// TIA Portal V16 export
// export: Created 2021-11-12T13:31:16.9009323Z, ExportSetting WithDefaults, DisplayName Totally Integrated Automation Portal, DisplayVersion V16 Update 3, DisplayName TIA Portal Version Control Interface, DisplayVersion V16 Update 2, DisplayName TIA Portal Openness, DisplayVersion V16 Update 3, DisplayName SINAMICS Startdrive Advanced, DisplayVersion V16 Update 5, DisplayName SINAMICS Startdrive G130, G150, S120, S150, SINAMICS MV, S210, DisplayVersion V16 Update 5, DisplayName SINAMICS Startdrive G110M, G120, G120C, G120D, G120P, G115D, DisplayVersion V16 Update 5, DisplayName STEP 7 Professional, DisplayVersion V16 Update 3, DisplayName STEP 7 Safety, DisplayVersion V16, DisplayName WinCC UA Professional, DisplayVersion V16 Update 3
FUNCTION_BLOCK "STD_Station"   // FB1101, LAD
TITLE = STD_Station
{ S7_Optimized_Access := 'TRUE' }
VERSION : 0.1
// Control of station - part of zone
// stored: AutoNumber false, IsIECCheckEnabled false, IsRetainMemResEnabled false, MemoryReserve 100, SetENOAutomatically false, UDAEnableTagReadback false
   VAR_INPUT
      IS_ZoneM : "UDT_Status_main";   // Status of zone
      IS_ZoneS : "UDT_Zone_Status_specific";   // Status of zone
      IB1StnExtCtrl : Bool;   // External control of station - own logic for automatic run
      IB1StnAutoRun : Bool;   // Station in automatic run mode - external signal
      IB1Rmt : Bool;   // Remote operation - operation from HMI panel
      IB1ManSwch : Bool;   // Switch in manual position
      IB1AutSwch : Bool;   // Switch in automatic position
      IB1SftyOK : Bool;   // Safety circuits ON
      IB1Run : Bool;   // Any device running
      IB1CollWrn : Bool;   // Any warning evaluated
      IB1CollErr : Bool;   // Any error evaluated
      IB1AllAutoRun : Bool;   // All drives in automatic run mode
      IB1AllEndOfCycle : Bool;   // All devices in end of cycle
      IB1AllEndOfProd : Bool;   // Production finished on all devices
      IB1AllInBasePos : Bool;   // All stations in base position
      IB1AllStopBefor : Bool;   // All stations stopped before operation
      IB1AllStopAfter : Bool;   // All stations stopped after finishing of operation
      IB1ReqBasePos : Bool;   // Request to move devices to base position
      IB1ReqEndOfCycle : Bool;   // Request for end of cycle
      IB1ReqEndOfProdAct : Bool;   // Request for end of production selection
      IB1ReqEndOfProdCncl : Bool;   // Request for end of production deselection
      IB1AutStartBtn : Bool;   // Button to start automatic
      IB1Stop : Bool;   // Command stop
      IB1Blink : Bool;   // Pulses for blinking
      IB1AlmSupp : Bool;   // Alarms suppressed
      II_DevSelNr : Int;   // Number of selected devices
   END_VAR
   VAR_OUTPUT
      OS_Status : Struct   // Output status
         Main : "UDT_Status_main";
         Specific : "UDT_Zone_Status_specific";
         Error : "UDT_Error01";
      END_STRUCT;
      OB1AutStart : Bool;   // LED for automatic start button
      OB1Man : Bool;   // LED for manual mode signalisation
      OB1Rmt : Bool;   // LED for remote control signalisation
      OB1SigAcs : Bool;   // Acoustic signalisation
   END_VAR
   VAR_IN_OUT
      XS_Parameter : "UDT_Station_Parameter";   // Parameters
      XS_Command : "UDT_Station_Command";   // Commands
   END_VAR
   VAR
      SS_Alarm : Struct   // Zone alarms
         Res_0_0 : Bool;
         Res_0_1 : Bool;
         Res_0_2 : Bool;
         Res_0_3 : Bool;
         Res_0_4 : Bool;
         Res_0_5 : Bool;
         Res_0_6 : Bool;
         Res_0_7 : Bool;
      END_STRUCT;
      SS_Warning : Struct   // Zone warnings
         EndOfCycle : Bool;   // End of cycle mode active / Konec cyklu aktivní / Mode de fin de cycle actif
         EndOfProd : Bool;   // End of production mode active / Konec produkce aktivní / Fin du mode de production actif
         StepMode : Bool;   // Step mode active / Krokový automat aktivní / Mode pas à pas actif
         StopBefor : Bool;   // Stop before operation active / Zastavení před procesem aktivní / Arrêtez avant l'opération actif
         StopAfter : Bool;   // Stop after operation active / Zastavení po procesu aktivní / Arrêter après l'opération actif
         BypasMode : Bool;   // Bypass mode active / Vynechání procesu aktivní / Mode bypass actif
         Res_0_6 : Bool;
         Res_0_7 : Bool;
      END_STRUCT;
      SB1AutoRun : Bool;   // Automatic operation started
      SB1AutoRunBasePos : Bool;   // Automatic operation - Run to base position
      SB1AutoRunProd : Bool;   // Automatic operation - Production
      SB1ModeAutStep : Bool;   // Mode automatic step selected
      SB1ModeStopBefor : Bool;   // Mode stop before production saelected
      SB1ModeStopAfter : Bool;   // Mode stop after production selected
      SB1ModeBypas : Bool;   // Mode bypass selected
      SB1ModeAut : Bool;   // Mode automatic
      SB1ModeMan : Bool;   // Mode manual
      SB1ModeOff : Bool;   // Mode off
      SB1ReqEndOfCycle : Bool;   // Request for end of cycle
      SB1ReqEndOfProd : Bool;   // Request for end of production
      SB1ManAutPE : Bool;   // Manual mode - positive edge
      SB1OffPE : Bool;   // Off mode - positive edge
      SB1ReqBasePosPE : Bool;   // Request for base position - positive edge
      SB1ReqEndOfCyclePE : Bool;   // Request end of cycle - positive edge
      SB1ReqEndOfProdActPE : Bool;   // Request end of production activation - positive edge
      SB1ReqEndOfProdCnclPE : Bool;   // Request end of production deactivation - positive edge
      SB1AutStart : Bool;   // Pulse start automatic sequence
      SB1AutStartAux : Bool;   // Auxiliary for start sequence
      SB1AuxHorn : Bool;   // To activate Horn before start
      SB1AutStartBtnPE : Bool;   // Automatic start 1 - positive edge
      ST_Horn { S7_SetPoint := 'True'} : TON_TIME;   // Timer for horn
      ST_Start { S7_SetPoint := 'True'} : TON_TIME;   // Timer to activate horn before start
      ST_AlmSupp { S7_SetPoint := 'True'} : IEC_TIMER;
   END_VAR
   VAR_TEMP
      TS_Status : Struct
         Main : "UDT_Status_main";
         Specific : "UDT_Zone_Status_specific";
         Error : "UDT_Error01";
      END_STRUCT;
      TS_Parameter : "UDT_Station_Parameter";   // Parameters
      TS_Command : "UDT_Station_Command";   // Commands
      TB1AlmSupp : Bool;
      TB1CollWrn : Bool;
      TB1ReqBasePosPE : Bool;   // Request for base position - positive edge
      TB1ReqEndOfCyclePE : Bool;   // Request end of cycle - positive edge
      TB1ReqEndOfProdActPE : Bool;   // Request end of production activation - positive edge
      TB1ReqEndOfProdCnclPE : Bool;   // Request end of production deactivation - positive edge
      TB1SigHorn : Bool;   // Horn before start signalisation
      TB1AutStartBtnPE : Bool;   // Automatic start 1 - positive edge
   END_VAR
   VAR CONSTANT
      CT_Horn : Time := T#2s;   // Time for horn before start
      CT_Start : Time := T#1s;   // Time for delay before start
      CT_AlmSupp : Time := T#3s;   // Time to delay alarm release
   END_VAR
   VAR_TEMP   // added for the SCL form of the ladder/FBD networks
      _w1 : Bool;
      _w2 : Bool;
   END_VAR
BEGIN

REGION Network 1: Clear temporary variables TS_Status - Main, Specific
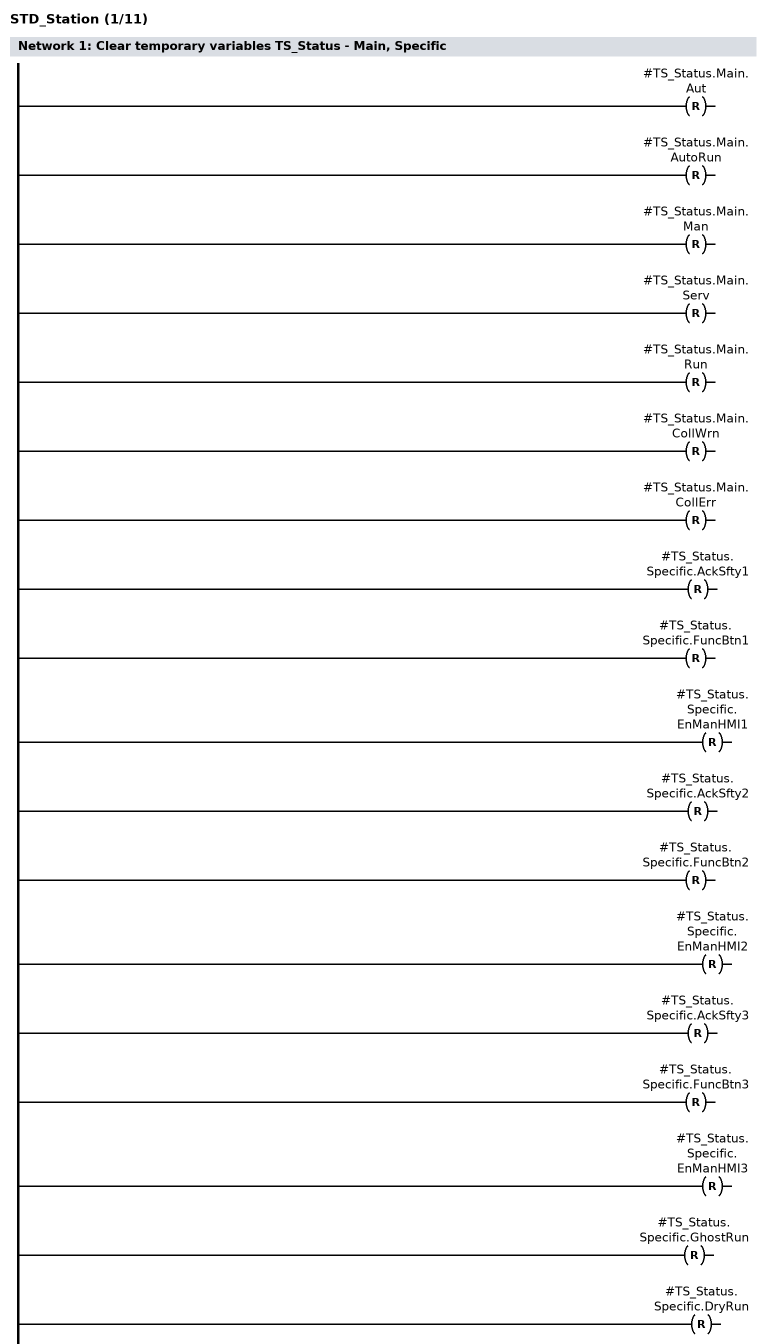
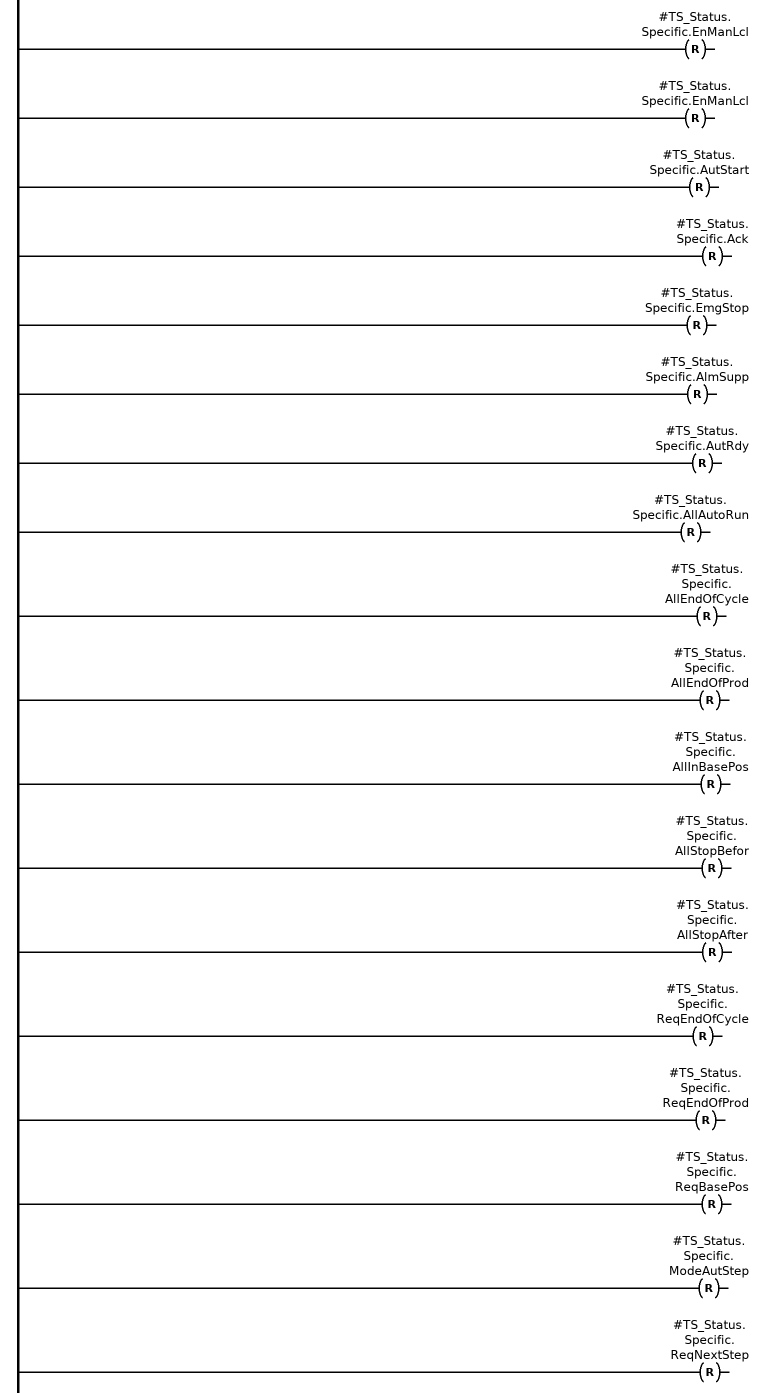
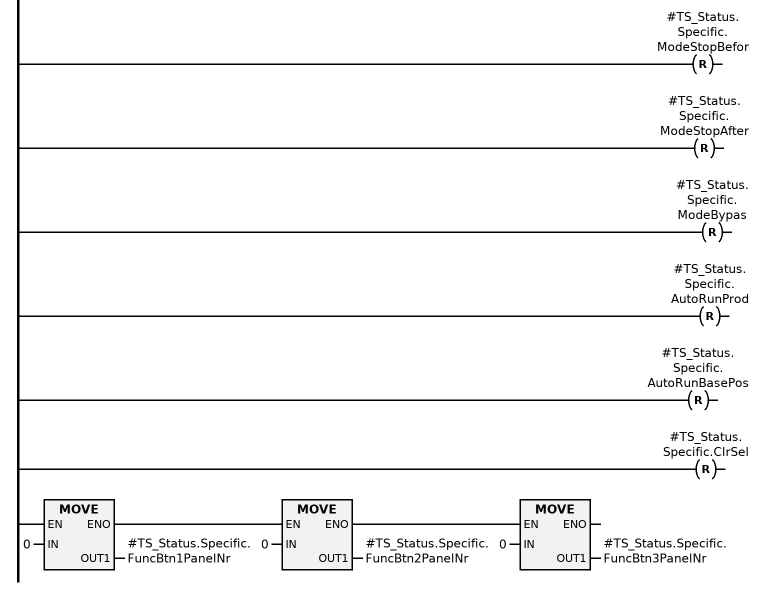
   RUNG wire#powerrail
      R_Coil( #TS_Status.Main.Aut )
   END_RUNG
   RUNG wire#powerrail
      R_Coil( #TS_Status.Main.AutoRun )
   END_RUNG
   RUNG wire#powerrail
      R_Coil( #TS_Status.Main.Man )
   END_RUNG
   RUNG wire#powerrail
      R_Coil( #TS_Status.Main.Serv )
   END_RUNG
   RUNG wire#powerrail
      R_Coil( #TS_Status.Main.Run )
   END_RUNG
   RUNG wire#powerrail
      R_Coil( #TS_Status.Main.CollWrn )
   END_RUNG
   RUNG wire#powerrail
      R_Coil( #TS_Status.Main.CollErr )
   END_RUNG
   RUNG wire#powerrail
      R_Coil( #TS_Status.Specific.AckSfty1 )
   END_RUNG
   RUNG wire#powerrail
      R_Coil( #TS_Status.Specific.FuncBtn1 )
   END_RUNG
   RUNG wire#powerrail
      R_Coil( #TS_Status.Specific.EnManHMI1 )
   END_RUNG
   RUNG wire#powerrail
      R_Coil( #TS_Status.Specific.AckSfty2 )
   END_RUNG
   RUNG wire#powerrail
      R_Coil( #TS_Status.Specific.FuncBtn2 )
   END_RUNG
   RUNG wire#powerrail
      R_Coil( #TS_Status.Specific.EnManHMI2 )
   END_RUNG
   RUNG wire#powerrail
      R_Coil( #TS_Status.Specific.AckSfty3 )
   END_RUNG
   RUNG wire#powerrail
      R_Coil( #TS_Status.Specific.FuncBtn3 )
   END_RUNG
   RUNG wire#powerrail
      R_Coil( #TS_Status.Specific.EnManHMI3 )
   END_RUNG
   RUNG wire#powerrail
      R_Coil( #TS_Status.Specific.GhostRun )
   END_RUNG
   RUNG wire#powerrail
      R_Coil( #TS_Status.Specific.DryRun )
   END_RUNG
   RUNG wire#powerrail
      R_Coil( #TS_Status.Specific.EnManLcl )
   END_RUNG
   RUNG wire#powerrail
      R_Coil( #TS_Status.Specific.EnManLcl )
   END_RUNG
   RUNG wire#powerrail
      R_Coil( #TS_Status.Specific.AutStart )
   END_RUNG
   RUNG wire#powerrail
      R_Coil( #TS_Status.Specific.Ack )
   END_RUNG
   RUNG wire#powerrail
      R_Coil( #TS_Status.Specific.EmgStop )
   END_RUNG
   RUNG wire#powerrail
      R_Coil( #TS_Status.Specific.AlmSupp )
   END_RUNG
   RUNG wire#powerrail
      R_Coil( #TS_Status.Specific.AutRdy )
   END_RUNG
   RUNG wire#powerrail
      R_Coil( #TS_Status.Specific.AllAutoRun )
   END_RUNG
   RUNG wire#powerrail
      R_Coil( #TS_Status.Specific.AllEndOfCycle )
   END_RUNG
   RUNG wire#powerrail
      R_Coil( #TS_Status.Specific.AllEndOfProd )
   END_RUNG
   RUNG wire#powerrail
      R_Coil( #TS_Status.Specific.AllInBasePos )
   END_RUNG
   RUNG wire#powerrail
      R_Coil( #TS_Status.Specific.AllStopBefor )
   END_RUNG
   RUNG wire#powerrail
      R_Coil( #TS_Status.Specific.AllStopAfter )
   END_RUNG
   RUNG wire#powerrail
      R_Coil( #TS_Status.Specific.ReqEndOfCycle )
   END_RUNG
   RUNG wire#powerrail
      R_Coil( #TS_Status.Specific.ReqEndOfProd )
   END_RUNG
   RUNG wire#powerrail
      R_Coil( #TS_Status.Specific.ReqBasePos )
   END_RUNG
   RUNG wire#powerrail
      R_Coil( #TS_Status.Specific.ModeAutStep )
   END_RUNG
   RUNG wire#powerrail
      R_Coil( #TS_Status.Specific.ReqNextStep )
   END_RUNG
   RUNG wire#powerrail
      R_Coil( #TS_Status.Specific.ModeStopBefor )
   END_RUNG
   RUNG wire#powerrail
      R_Coil( #TS_Status.Specific.ModeStopAfter )
   END_RUNG
   RUNG wire#powerrail
      R_Coil( #TS_Status.Specific.ModeBypas )
   END_RUNG
   RUNG wire#powerrail
      R_Coil( #TS_Status.Specific.AutoRunProd )
   END_RUNG
   RUNG wire#powerrail
      R_Coil( #TS_Status.Specific.AutoRunBasePos )
   END_RUNG
   RUNG wire#powerrail
      R_Coil( #TS_Status.Specific.ClrSel )
   END_RUNG
   RUNG wire#powerrail
      { S7_GenerateENO := "TRUE" } Move(in := 0, out1 => #TS_Status.Specific.FuncBtn1PanelNr)
      { S7_GenerateENO := "TRUE" } Move(in := 0, out1 => #TS_Status.Specific.FuncBtn2PanelNr)
      { S7_GenerateENO := "TRUE" } Move(in := 0, out1 => #TS_Status.Specific.FuncBtn3PanelNr)
   END_RUNG
   // the same network as SCL:
   // ENO of a box is taken as its EN; it also drops when the box reports an error
   #TS_Status.Main.Aut := FALSE;
   #TS_Status.Main.AutoRun := FALSE;
   #TS_Status.Main.Man := FALSE;
   #TS_Status.Main.Serv := FALSE;
   #TS_Status.Main.Run := FALSE;
   #TS_Status.Main.CollWrn := FALSE;
   #TS_Status.Main.CollErr := FALSE;
   #TS_Status.Specific.AckSfty1 := FALSE;
   #TS_Status.Specific.FuncBtn1 := FALSE;
   #TS_Status.Specific.EnManHMI1 := FALSE;
   #TS_Status.Specific.AckSfty2 := FALSE;
   #TS_Status.Specific.FuncBtn2 := FALSE;
   #TS_Status.Specific.EnManHMI2 := FALSE;
   #TS_Status.Specific.AckSfty3 := FALSE;
   #TS_Status.Specific.FuncBtn3 := FALSE;
   #TS_Status.Specific.EnManHMI3 := FALSE;
   #TS_Status.Specific.GhostRun := FALSE;
   #TS_Status.Specific.DryRun := FALSE;
   #TS_Status.Specific.EnManLcl := FALSE;
   #TS_Status.Specific.EnManLcl := FALSE;
   #TS_Status.Specific.AutStart := FALSE;
   #TS_Status.Specific.Ack := FALSE;
   #TS_Status.Specific.EmgStop := FALSE;
   #TS_Status.Specific.AlmSupp := FALSE;
   #TS_Status.Specific.AutRdy := FALSE;
   #TS_Status.Specific.AllAutoRun := FALSE;
   #TS_Status.Specific.AllEndOfCycle := FALSE;
   #TS_Status.Specific.AllEndOfProd := FALSE;
   #TS_Status.Specific.AllInBasePos := FALSE;
   #TS_Status.Specific.AllStopBefor := FALSE;
   #TS_Status.Specific.AllStopAfter := FALSE;
   #TS_Status.Specific.ReqEndOfCycle := FALSE;
   #TS_Status.Specific.ReqEndOfProd := FALSE;
   #TS_Status.Specific.ReqBasePos := FALSE;
   #TS_Status.Specific.ModeAutStep := FALSE;
   #TS_Status.Specific.ReqNextStep := FALSE;
   #TS_Status.Specific.ModeStopBefor := FALSE;
   #TS_Status.Specific.ModeStopAfter := FALSE;
   #TS_Status.Specific.ModeBypas := FALSE;
   #TS_Status.Specific.AutoRunProd := FALSE;
   #TS_Status.Specific.AutoRunBasePos := FALSE;
   #TS_Status.Specific.ClrSel := FALSE;
   #TS_Status.Specific.FuncBtn1PanelNr := 0;
   #TS_Status.Specific.FuncBtn2PanelNr := 0;
   #TS_Status.Specific.FuncBtn3PanelNr := 0;
END_REGION

REGION Network 2: Copy In/Out variables to temporary variables
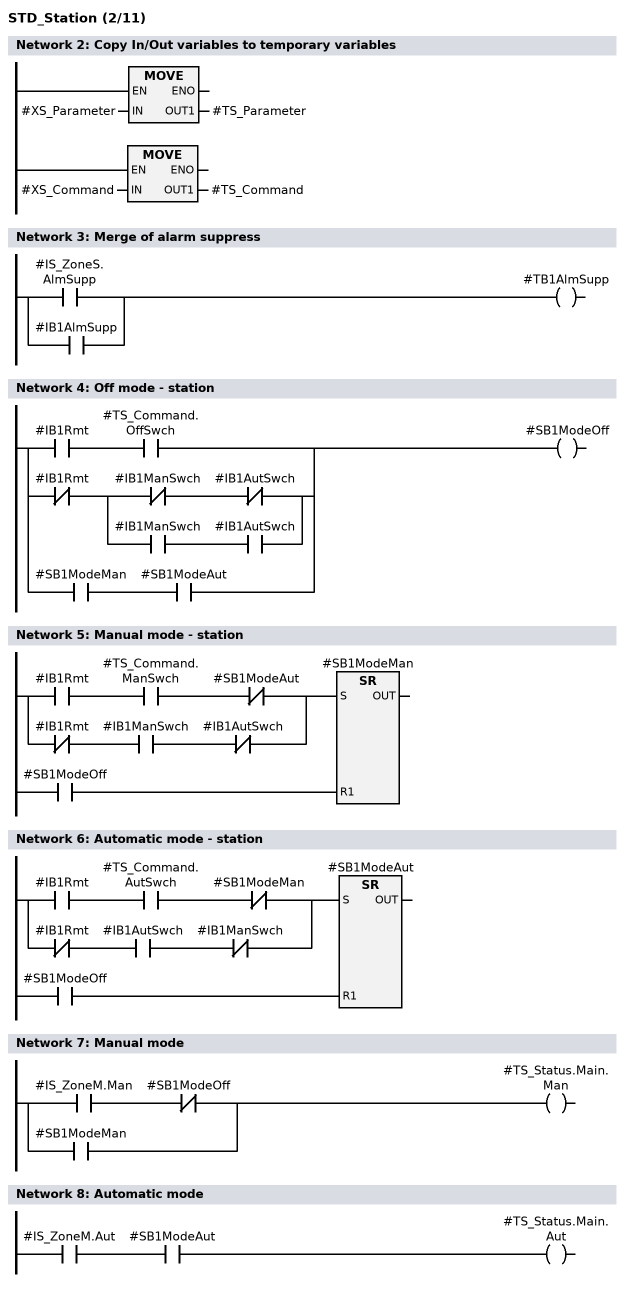
   RUNG wire#powerrail
      { S7_GenerateENO := "TRUE" } Move(in := #XS_Parameter, out1 => #TS_Parameter)
   END_RUNG
   RUNG wire#powerrail
      { S7_GenerateENO := "TRUE" } Move(in := #XS_Command, out1 => #TS_Command)
   END_RUNG
   // the same network as SCL:
   #TS_Parameter := #XS_Parameter;
   #TS_Command := #XS_Command;
END_REGION

REGION Network 3: Merge of alarm suppress
   RUNG wire#powerrail
      Contact( #IS_ZoneS.AlmSupp )
      wire#w1
      Coil( #TB1AlmSupp )
   END_RUNG
   RUNG wire#powerrail
      Contact( #IB1AlmSupp )
   END_RUNG wire#w1
   // the same network as SCL:
   #TB1AlmSupp := #IS_ZoneS.AlmSupp OR #IB1AlmSupp;
END_REGION

REGION Network 4: Off mode - station
   RUNG wire#powerrail
      Contact( #IB1Rmt )
      Contact( #TS_Command.OffSwch )
      wire#w1
      Coil( #SB1ModeOff )
   END_RUNG
   RUNG wire#powerrail
      I_Contact( #IB1Rmt )
      wire#w2
      I_Contact( #IB1ManSwch )
      I_Contact( #IB1AutSwch )
   END_RUNG wire#w1
   RUNG wire#w2
      Contact( #IB1ManSwch )
      Contact( #IB1AutSwch )
   END_RUNG wire#w1
   RUNG wire#powerrail
      Contact( #SB1ModeMan )
      Contact( #SB1ModeAut )
   END_RUNG wire#w1
   // the same network as SCL:
   #SB1ModeOff := (#IB1Rmt AND #TS_Command.OffSwch) OR (NOT #IB1Rmt AND ((NOT #IB1ManSwch AND NOT #IB1AutSwch) OR (#IB1ManSwch AND #IB1AutSwch))) OR (#SB1ModeMan AND #SB1ModeAut);
END_REGION

REGION Network 5: Manual mode - station
   RUNG wire#powerrail
      Contact( #IB1Rmt )
      Contact( #TS_Command.ManSwch )
      I_Contact( #SB1ModeAut )
      wire#w1
      S_SR(operand := #SB1ModeMan, r1 := wire#w2)
   END_RUNG
   RUNG wire#powerrail
      I_Contact( #IB1Rmt )
      Contact( #IB1ManSwch )
      I_Contact( #IB1AutSwch )
   END_RUNG wire#w1
   RUNG wire#powerrail
      Contact( #SB1ModeOff )
   END_RUNG wire#w2
   // the same network as SCL:
   IF (#IB1Rmt AND #TS_Command.ManSwch AND NOT #SB1ModeAut) OR (NOT #IB1Rmt AND #IB1ManSwch AND NOT #IB1AutSwch) THEN
       #SB1ModeMan := TRUE;   // SR flip-flop
   END_IF;
   IF #SB1ModeOff THEN #SB1ModeMan := FALSE; END_IF;
END_REGION

REGION Network 6: Automatic mode - station
   RUNG wire#powerrail
      Contact( #IB1Rmt )
      Contact( #TS_Command.AutSwch )
      I_Contact( #SB1ModeMan )
      wire#w1
      S_SR(operand := #SB1ModeAut, r1 := wire#w2)
   END_RUNG
   RUNG wire#powerrail
      I_Contact( #IB1Rmt )
      Contact( #IB1AutSwch )
      I_Contact( #IB1ManSwch )
   END_RUNG wire#w1
   RUNG wire#powerrail
      Contact( #SB1ModeOff )
   END_RUNG wire#w2
   // the same network as SCL:
   IF (#IB1Rmt AND #TS_Command.AutSwch AND NOT #SB1ModeMan) OR (NOT #IB1Rmt AND #IB1AutSwch AND NOT #IB1ManSwch) THEN
       #SB1ModeAut := TRUE;   // SR flip-flop
   END_IF;
   IF #SB1ModeOff THEN #SB1ModeAut := FALSE; END_IF;
END_REGION

REGION Network 7: Manual mode
   RUNG wire#powerrail
      Contact( #IS_ZoneM.Man )
      I_Contact( #SB1ModeOff )
      wire#w1
      Coil( #TS_Status.Main.Man )
   END_RUNG
   RUNG wire#powerrail
      Contact( #SB1ModeMan )
   END_RUNG wire#w1
   // the same network as SCL:
   #TS_Status.Main.Man := (#IS_ZoneM.Man AND NOT #SB1ModeOff) OR #SB1ModeMan;
END_REGION

REGION Network 8: Automatic mode
   RUNG wire#powerrail
      Contact( #IS_ZoneM.Aut )
      Contact( #SB1ModeAut )
      Coil( #TS_Status.Main.Aut )
   END_RUNG
   // the same network as SCL:
   #TS_Status.Main.Aut := #IS_ZoneM.Aut AND #SB1ModeAut;
END_REGION

REGION Network 9: Automatic start - pulse
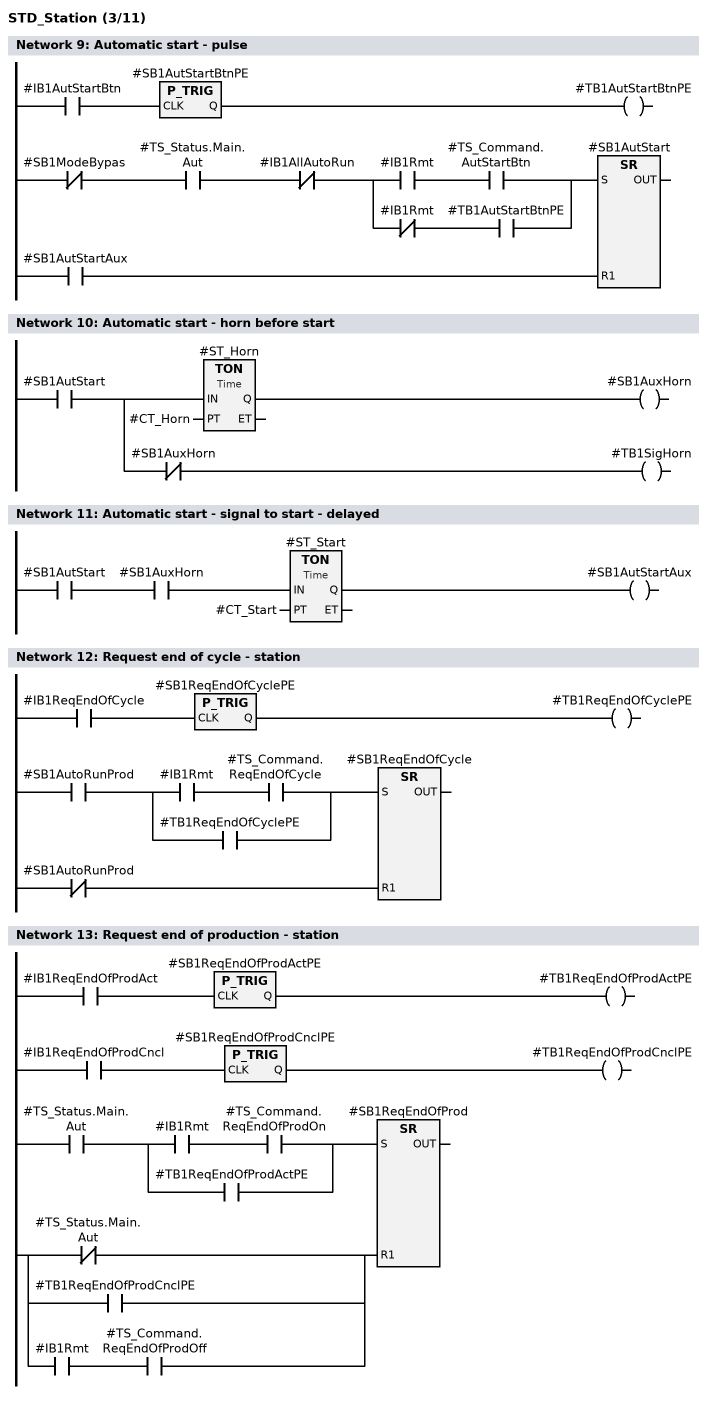
   RUNG wire#powerrail
      Contact( #IB1AutStartBtn )
      P_Trig( #SB1AutStartBtnPE )
      Coil( #TB1AutStartBtnPE )
   END_RUNG
   RUNG wire#powerrail
      I_Contact( #SB1ModeBypas )
      Contact( #TS_Status.Main.Aut )
      I_Contact( #IB1AllAutoRun )
      wire#w1
      Contact( #IB1Rmt )
      Contact( #TS_Command.AutStartBtn )
      wire#w2
      S_SR(operand := #SB1AutStart, r1 := wire#w3)
   END_RUNG
   RUNG wire#w1
      I_Contact( #IB1Rmt )
      Contact( #TB1AutStartBtnPE )
   END_RUNG wire#w2
   RUNG wire#powerrail
      Contact( #SB1AutStartAux )
   END_RUNG wire#w3
   // the same network as SCL:
   #_w1 := #IB1AutStartBtn AND NOT #SB1AutStartBtnPE;   // rising edge
   #SB1AutStartBtnPE := #IB1AutStartBtn;
   #TB1AutStartBtnPE := #_w1;
   IF NOT #SB1ModeBypas AND #TS_Status.Main.Aut AND NOT #IB1AllAutoRun AND ((#IB1Rmt AND #TS_Command.AutStartBtn) OR (NOT #IB1Rmt AND #TB1AutStartBtnPE)) THEN
       #SB1AutStart := TRUE;   // SR flip-flop
   END_IF;
   IF #SB1AutStartAux THEN #SB1AutStart := FALSE; END_IF;
END_REGION

REGION Network 10: Automatic start - horn before start
   RUNG wire#powerrail
      Contact( #SB1AutStart )
      wire#w1
      { S7_Templates := "time_type := Time" } #ST_Horn.TON(pt := #CT_Horn, et =>)
      Coil( #SB1AuxHorn )
   END_RUNG
   RUNG wire#w1
      I_Contact( #SB1AuxHorn )
      Coil( #TB1SigHorn )
   END_RUNG
   // the same network as SCL:
   #ST_Horn(IN := #SB1AutStart, PT := #CT_Horn);   // TON
   #SB1AuxHorn := #ST_Horn.Q;
   #TB1SigHorn := #SB1AutStart AND NOT #SB1AuxHorn;
END_REGION

REGION Network 11: Automatic start - signal to start - delayed
   RUNG wire#powerrail
      Contact( #SB1AutStart )
      Contact( #SB1AuxHorn )
      { S7_Templates := "time_type := Time" } #ST_Start.TON(pt := #CT_Start, et =>)
      Coil( #SB1AutStartAux )
   END_RUNG
   // the same network as SCL:
   #ST_Start(IN := #SB1AutStart AND #SB1AuxHorn, PT := #CT_Start);   // TON
   #SB1AutStartAux := #ST_Start.Q;
END_REGION

REGION Network 12: Request end of cycle - station
   RUNG wire#powerrail
      Contact( #IB1ReqEndOfCycle )
      P_Trig( #SB1ReqEndOfCyclePE )
      Coil( #TB1ReqEndOfCyclePE )
   END_RUNG
   RUNG wire#powerrail
      Contact( #SB1AutoRunProd )
      wire#w1
      Contact( #IB1Rmt )
      Contact( #TS_Command.ReqEndOfCycle )
      wire#w2
      S_SR(operand := #SB1ReqEndOfCycle, r1 := wire#w3)
   END_RUNG
   RUNG wire#w1
      Contact( #TB1ReqEndOfCyclePE )
   END_RUNG wire#w2
   RUNG wire#powerrail
      I_Contact( #SB1AutoRunProd )
   END_RUNG wire#w3
   // the same network as SCL:
   #_w1 := #IB1ReqEndOfCycle AND NOT #SB1ReqEndOfCyclePE;   // rising edge
   #SB1ReqEndOfCyclePE := #IB1ReqEndOfCycle;
   #TB1ReqEndOfCyclePE := #_w1;
   IF #SB1AutoRunProd AND ((#IB1Rmt AND #TS_Command.ReqEndOfCycle) OR #TB1ReqEndOfCyclePE) THEN
       #SB1ReqEndOfCycle := TRUE;   // SR flip-flop
   END_IF;
   IF NOT #SB1AutoRunProd THEN #SB1ReqEndOfCycle := FALSE; END_IF;
END_REGION

REGION Network 13: Request end of production - station
   RUNG wire#powerrail
      Contact( #IB1ReqEndOfProdAct )
      P_Trig( #SB1ReqEndOfProdActPE )
      Coil( #TB1ReqEndOfProdActPE )
   END_RUNG
   RUNG wire#powerrail
      Contact( #IB1ReqEndOfProdCncl )
      P_Trig( #SB1ReqEndOfProdCnclPE )
      Coil( #TB1ReqEndOfProdCnclPE )
   END_RUNG
   RUNG wire#powerrail
      Contact( #TS_Status.Main.Aut )
      wire#w1
      Contact( #IB1Rmt )
      Contact( #TS_Command.ReqEndOfProdOn )
      wire#w2
      S_SR(operand := #SB1ReqEndOfProd, r1 := wire#w3)
   END_RUNG
   RUNG wire#w1
      Contact( #TB1ReqEndOfProdActPE )
   END_RUNG wire#w2
   RUNG wire#powerrail
      I_Contact( #TS_Status.Main.Aut )
   END_RUNG wire#w3
   RUNG wire#powerrail
      Contact( #TB1ReqEndOfProdCnclPE )
   END_RUNG wire#w3
   RUNG wire#powerrail
      Contact( #IB1Rmt )
      Contact( #TS_Command.ReqEndOfProdOff )
   END_RUNG wire#w3
   // the same network as SCL:
   #_w1 := #IB1ReqEndOfProdAct AND NOT #SB1ReqEndOfProdActPE;   // rising edge
   #SB1ReqEndOfProdActPE := #IB1ReqEndOfProdAct;
   #TB1ReqEndOfProdActPE := #_w1;
   #_w2 := #IB1ReqEndOfProdCncl AND NOT #SB1ReqEndOfProdCnclPE;   // rising edge
   #SB1ReqEndOfProdCnclPE := #IB1ReqEndOfProdCncl;
   #TB1ReqEndOfProdCnclPE := #_w2;
   IF #TS_Status.Main.Aut AND ((#IB1Rmt AND #TS_Command.ReqEndOfProdOn) OR #TB1ReqEndOfProdActPE) THEN
       #SB1ReqEndOfProd := TRUE;   // SR flip-flop
   END_IF;
   IF NOT #TS_Status.Main.Aut OR #TB1ReqEndOfProdCnclPE OR (#IB1Rmt AND #TS_Command.ReqEndOfProdOff) THEN
       #SB1ReqEndOfProd := FALSE;
   END_IF;
END_REGION

REGION Network 14: Request end of cycle
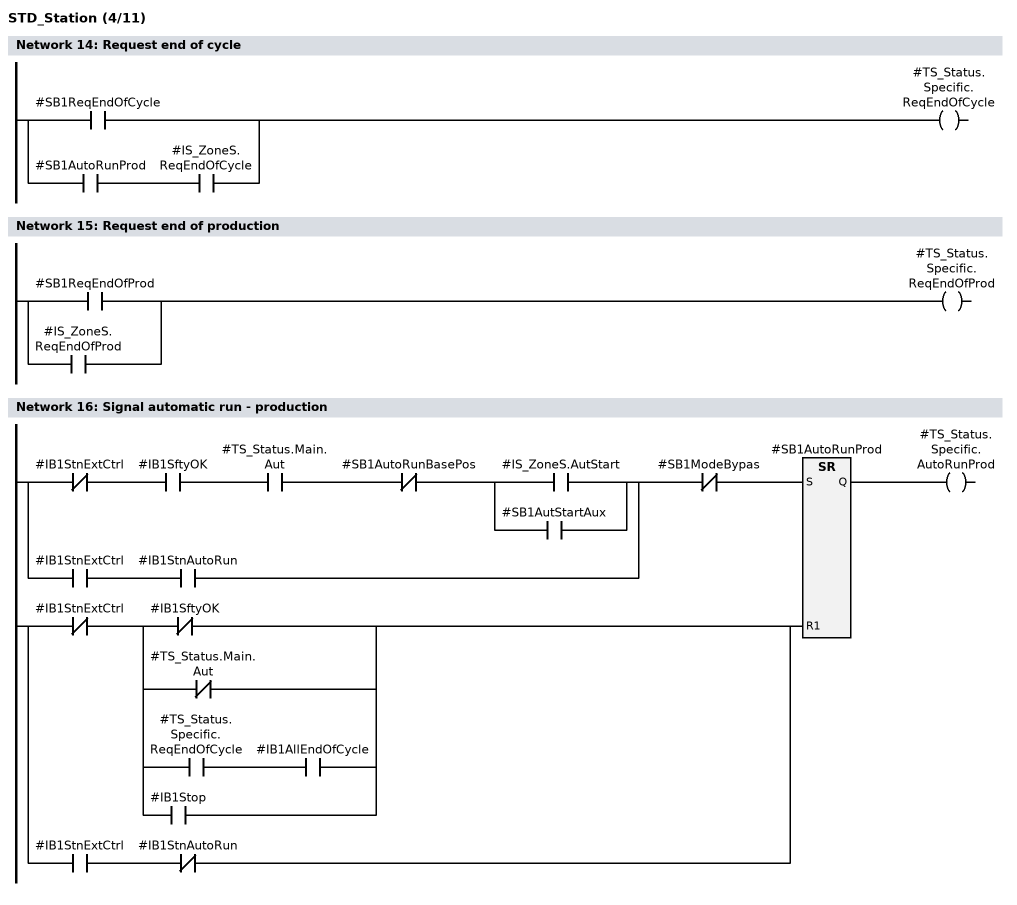
   RUNG wire#powerrail
      Contact( #SB1ReqEndOfCycle )
      wire#w1
      Coil( #TS_Status.Specific.ReqEndOfCycle )
   END_RUNG
   RUNG wire#powerrail
      Contact( #SB1AutoRunProd )
      Contact( #IS_ZoneS.ReqEndOfCycle )
   END_RUNG wire#w1
   // the same network as SCL:
   #TS_Status.Specific.ReqEndOfCycle := #SB1ReqEndOfCycle OR (#SB1AutoRunProd AND #IS_ZoneS.ReqEndOfCycle);
END_REGION

REGION Network 15: Request end of production
   RUNG wire#powerrail
      Contact( #SB1ReqEndOfProd )
      wire#w1
      Coil( #TS_Status.Specific.ReqEndOfProd )
   END_RUNG
   RUNG wire#powerrail
      Contact( #IS_ZoneS.ReqEndOfProd )
   END_RUNG wire#w1
   // the same network as SCL:
   #TS_Status.Specific.ReqEndOfProd := #SB1ReqEndOfProd OR #IS_ZoneS.ReqEndOfProd;
END_REGION

REGION Network 16: Signal automatic run - production
   RUNG wire#powerrail
      I_Contact( #IB1StnExtCtrl )
      Contact( #IB1SftyOK )
      Contact( #TS_Status.Main.Aut )
      I_Contact( #SB1AutoRunBasePos )
      wire#w1
      Contact( #IS_ZoneS.AutStart )
      wire#w2
      I_Contact( #SB1ModeBypas )
      S_SR(operand := #SB1AutoRunProd, r1 := wire#w4)
      Coil( #TS_Status.Specific.AutoRunProd )
   END_RUNG
   RUNG wire#w1
      Contact( #SB1AutStartAux )
   END_RUNG wire#w2
   RUNG wire#powerrail
      Contact( #IB1StnExtCtrl )
      Contact( #IB1StnAutoRun )
   END_RUNG wire#w2
   RUNG wire#powerrail
      I_Contact( #IB1StnExtCtrl )
      wire#w3
      I_Contact( #IB1SftyOK )
   END_RUNG wire#w4
   RUNG wire#w3
      I_Contact( #TS_Status.Main.Aut )
   END_RUNG wire#w4
   RUNG wire#w3
      Contact( #TS_Status.Specific.ReqEndOfCycle )
      Contact( #IB1AllEndOfCycle )
   END_RUNG wire#w4
   RUNG wire#w3
      Contact( #IB1Stop )
   END_RUNG wire#w4
   RUNG wire#powerrail
      Contact( #IB1StnExtCtrl )
      I_Contact( #IB1StnAutoRun )
   END_RUNG wire#w4
   // the same network as SCL:
   IF ((NOT #IB1StnExtCtrl AND #IB1SftyOK AND #TS_Status.Main.Aut AND NOT #SB1AutoRunBasePos AND (#IS_ZoneS.AutStart OR #SB1AutStartAux)) OR (#IB1StnExtCtrl AND #IB1StnAutoRun)) AND NOT #SB1ModeBypas THEN
       #SB1AutoRunProd := TRUE;   // SR flip-flop
   END_IF;
   IF (NOT #IB1StnExtCtrl AND (NOT #IB1SftyOK OR NOT #TS_Status.Main.Aut OR (#TS_Status.Specific.ReqEndOfCycle AND #IB1AllEndOfCycle) OR #IB1Stop)) OR (#IB1StnExtCtrl AND NOT #IB1StnAutoRun) THEN
       #SB1AutoRunProd := FALSE;
   END_IF;
   #TS_Status.Specific.AutoRunProd := #SB1AutoRunProd;
END_REGION

REGION Network 17: Signal automatic run - base position
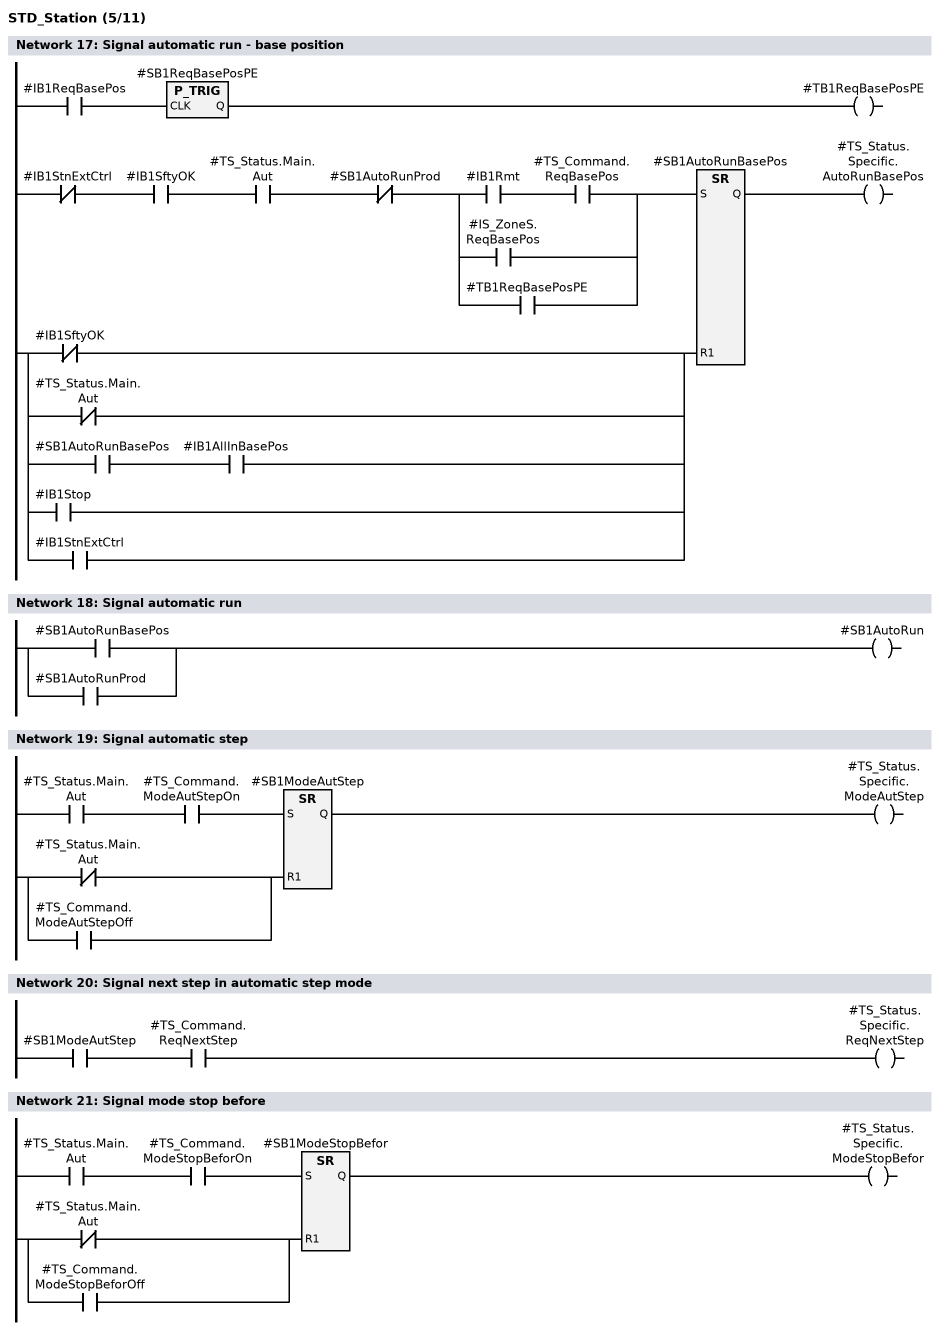
   RUNG wire#powerrail
      Contact( #IB1ReqBasePos )
      P_Trig( #SB1ReqBasePosPE )
      Coil( #TB1ReqBasePosPE )
   END_RUNG
   RUNG wire#powerrail
      I_Contact( #IB1StnExtCtrl )
      Contact( #IB1SftyOK )
      Contact( #TS_Status.Main.Aut )
      I_Contact( #SB1AutoRunProd )
      wire#w1
      Contact( #IB1Rmt )
      Contact( #TS_Command.ReqBasePos )
      wire#w2
      S_SR(operand := #SB1AutoRunBasePos, r1 := wire#w3)
      Coil( #TS_Status.Specific.AutoRunBasePos )
   END_RUNG
   RUNG wire#w1
      Contact( #IS_ZoneS.ReqBasePos )
   END_RUNG wire#w2
   RUNG wire#w1
      Contact( #TB1ReqBasePosPE )
   END_RUNG wire#w2
   RUNG wire#powerrail
      I_Contact( #IB1SftyOK )
   END_RUNG wire#w3
   RUNG wire#powerrail
      I_Contact( #TS_Status.Main.Aut )
   END_RUNG wire#w3
   RUNG wire#powerrail
      Contact( #SB1AutoRunBasePos )
      Contact( #IB1AllInBasePos )
   END_RUNG wire#w3
   RUNG wire#powerrail
      Contact( #IB1Stop )
   END_RUNG wire#w3
   RUNG wire#powerrail
      Contact( #IB1StnExtCtrl )
   END_RUNG wire#w3
   // the same network as SCL:
   #_w1 := #IB1ReqBasePos AND NOT #SB1ReqBasePosPE;   // rising edge
   #SB1ReqBasePosPE := #IB1ReqBasePos;
   #TB1ReqBasePosPE := #_w1;
   #_w2 := NOT #IB1SftyOK OR NOT #TS_Status.Main.Aut OR (#SB1AutoRunBasePos AND #IB1AllInBasePos) OR #IB1Stop OR #IB1StnExtCtrl;
   IF NOT #IB1StnExtCtrl AND #IB1SftyOK AND #TS_Status.Main.Aut AND NOT #SB1AutoRunProd AND ((#IB1Rmt AND #TS_Command.ReqBasePos) OR #IS_ZoneS.ReqBasePos OR #TB1ReqBasePosPE) THEN
       #SB1AutoRunBasePos := TRUE;   // SR flip-flop
   END_IF;
   IF #_w2 THEN #SB1AutoRunBasePos := FALSE; END_IF;
   #TS_Status.Specific.AutoRunBasePos := #SB1AutoRunBasePos;
END_REGION

REGION Network 18: Signal automatic run
   RUNG wire#powerrail
      Contact( #SB1AutoRunBasePos )
      wire#w1
      Coil( #SB1AutoRun )
   END_RUNG
   RUNG wire#powerrail
      Contact( #SB1AutoRunProd )
   END_RUNG wire#w1
   // the same network as SCL:
   #SB1AutoRun := #SB1AutoRunBasePos OR #SB1AutoRunProd;
END_REGION

REGION Network 19: Signal automatic step
   RUNG wire#powerrail
      Contact( #TS_Status.Main.Aut )
      Contact( #TS_Command.ModeAutStepOn )
      S_SR(operand := #SB1ModeAutStep, r1 := wire#w1)
      Coil( #TS_Status.Specific.ModeAutStep )
   END_RUNG
   RUNG wire#powerrail
      I_Contact( #TS_Status.Main.Aut )
   END_RUNG wire#w1
   RUNG wire#powerrail
      Contact( #TS_Command.ModeAutStepOff )
   END_RUNG wire#w1
   // the same network as SCL:
   IF #TS_Status.Main.Aut AND #TS_Command.ModeAutStepOn THEN
       #SB1ModeAutStep := TRUE;   // SR flip-flop
   END_IF;
   IF NOT #TS_Status.Main.Aut OR #TS_Command.ModeAutStepOff THEN #SB1ModeAutStep := FALSE; END_IF;
   #TS_Status.Specific.ModeAutStep := #SB1ModeAutStep;
END_REGION

REGION Network 20: Signal next step in automatic step mode
   RUNG wire#powerrail
      Contact( #SB1ModeAutStep )
      Contact( #TS_Command.ReqNextStep )
      Coil( #TS_Status.Specific.ReqNextStep )
   END_RUNG
   // the same network as SCL:
   #TS_Status.Specific.ReqNextStep := #SB1ModeAutStep AND #TS_Command.ReqNextStep;
END_REGION

REGION Network 21: Signal mode stop before
   RUNG wire#powerrail
      Contact( #TS_Status.Main.Aut )
      Contact( #TS_Command.ModeStopBeforOn )
      S_SR(operand := #SB1ModeStopBefor, r1 := wire#w1)
      Coil( #TS_Status.Specific.ModeStopBefor )
   END_RUNG
   RUNG wire#powerrail
      I_Contact( #TS_Status.Main.Aut )
   END_RUNG wire#w1
   RUNG wire#powerrail
      Contact( #TS_Command.ModeStopBeforOff )
   END_RUNG wire#w1
   // the same network as SCL:
   IF #TS_Status.Main.Aut AND #TS_Command.ModeStopBeforOn THEN
       #SB1ModeStopBefor := TRUE;   // SR flip-flop
   END_IF;
   IF NOT #TS_Status.Main.Aut OR #TS_Command.ModeStopBeforOff THEN #SB1ModeStopBefor := FALSE; END_IF;
   #TS_Status.Specific.ModeStopBefor := #SB1ModeStopBefor;
END_REGION

REGION Network 22: Signal mode stop after
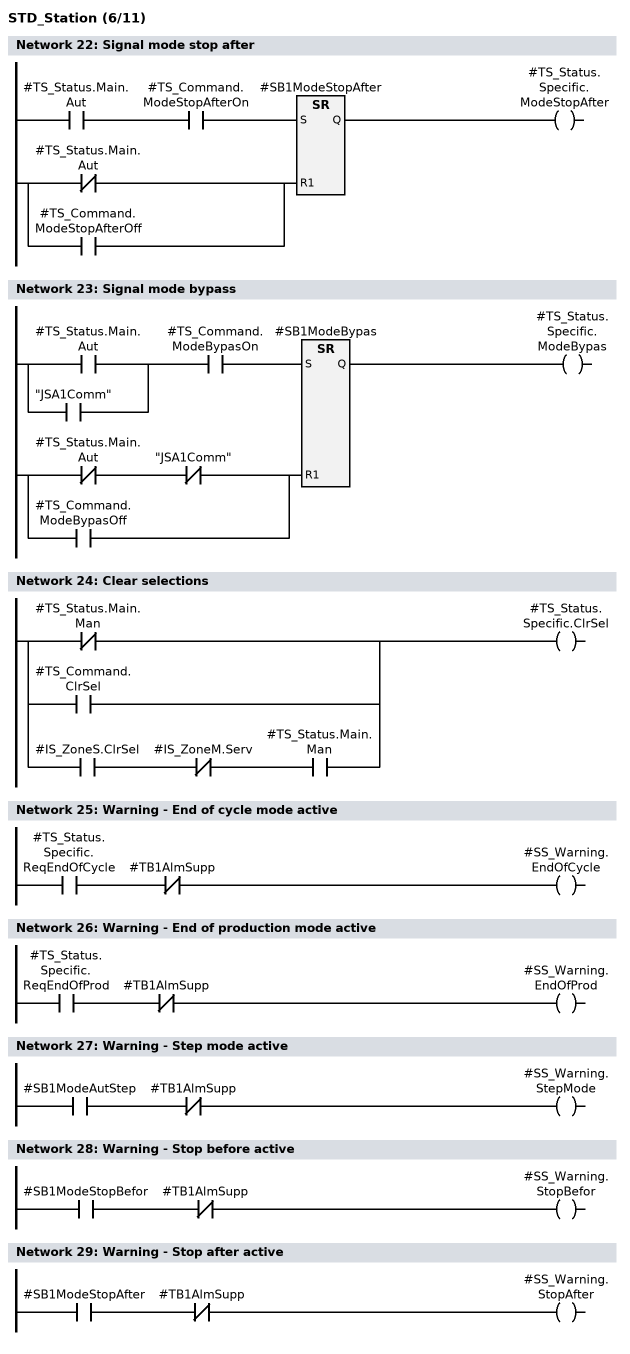
   RUNG wire#powerrail
      Contact( #TS_Status.Main.Aut )
      Contact( #TS_Command.ModeStopAfterOn )
      S_SR(operand := #SB1ModeStopAfter, r1 := wire#w1)
      Coil( #TS_Status.Specific.ModeStopAfter )
   END_RUNG
   RUNG wire#powerrail
      I_Contact( #TS_Status.Main.Aut )
   END_RUNG wire#w1
   RUNG wire#powerrail
      Contact( #TS_Command.ModeStopAfterOff )
   END_RUNG wire#w1
   // the same network as SCL:
   IF #TS_Status.Main.Aut AND #TS_Command.ModeStopAfterOn THEN
       #SB1ModeStopAfter := TRUE;   // SR flip-flop
   END_IF;
   IF NOT #TS_Status.Main.Aut OR #TS_Command.ModeStopAfterOff THEN #SB1ModeStopAfter := FALSE; END_IF;
   #TS_Status.Specific.ModeStopAfter := #SB1ModeStopAfter;
END_REGION

REGION Network 23: Signal mode bypass
   RUNG wire#powerrail
      Contact( #TS_Status.Main.Aut )
      wire#w1
      Contact( #TS_Command.ModeBypasOn )
      S_SR(operand := #SB1ModeBypas, r1 := wire#w2)
      Coil( #TS_Status.Specific.ModeBypas )
   END_RUNG
   RUNG wire#powerrail
      Contact( "JSA1Comm" )
   END_RUNG wire#w1
   RUNG wire#powerrail
      I_Contact( #TS_Status.Main.Aut )
      I_Contact( "JSA1Comm" )
   END_RUNG wire#w2
   RUNG wire#powerrail
      Contact( #TS_Command.ModeBypasOff )
   END_RUNG wire#w2
   // the same network as SCL:
   IF (#TS_Status.Main.Aut OR "JSA1Comm") AND #TS_Command.ModeBypasOn THEN
       #SB1ModeBypas := TRUE;   // SR flip-flop
   END_IF;
   IF (NOT #TS_Status.Main.Aut AND NOT "JSA1Comm") OR #TS_Command.ModeBypasOff THEN
       #SB1ModeBypas := FALSE;
   END_IF;
   #TS_Status.Specific.ModeBypas := #SB1ModeBypas;
END_REGION

REGION Network 24: Clear selections
   RUNG wire#powerrail
      I_Contact( #TS_Status.Main.Man )
      wire#w1
      Coil( #TS_Status.Specific.ClrSel )
   END_RUNG
   RUNG wire#powerrail
      Contact( #TS_Command.ClrSel )
   END_RUNG wire#w1
   RUNG wire#powerrail
      Contact( #IS_ZoneS.ClrSel )
      I_Contact( #IS_ZoneM.Serv )
      Contact( #TS_Status.Main.Man )
   END_RUNG wire#w1
   // the same network as SCL:
   #TS_Status.Specific.ClrSel := NOT #TS_Status.Main.Man OR #TS_Command.ClrSel OR (#IS_ZoneS.ClrSel AND NOT #IS_ZoneM.Serv AND #TS_Status.Main.Man);
END_REGION

REGION Network 25: Warning - End of cycle mode active
   RUNG wire#powerrail
      Contact( #TS_Status.Specific.ReqEndOfCycle )
      I_Contact( #TB1AlmSupp )
      Coil( #SS_Warning.EndOfCycle )
   END_RUNG
   // the same network as SCL:
   #SS_Warning.EndOfCycle := #TS_Status.Specific.ReqEndOfCycle AND NOT #TB1AlmSupp;
END_REGION

REGION Network 26: Warning - End of production mode active
   RUNG wire#powerrail
      Contact( #TS_Status.Specific.ReqEndOfProd )
      I_Contact( #TB1AlmSupp )
      Coil( #SS_Warning.EndOfProd )
   END_RUNG
   // the same network as SCL:
   #SS_Warning.EndOfProd := #TS_Status.Specific.ReqEndOfProd AND NOT #TB1AlmSupp;
END_REGION

REGION Network 27: Warning - Step mode active
   RUNG wire#powerrail
      Contact( #SB1ModeAutStep )
      I_Contact( #TB1AlmSupp )
      Coil( #SS_Warning.StepMode )
   END_RUNG
   // the same network as SCL:
   #SS_Warning.StepMode := #SB1ModeAutStep AND NOT #TB1AlmSupp;
END_REGION

REGION Network 28: Warning - Stop before active
   RUNG wire#powerrail
      Contact( #SB1ModeStopBefor )
      I_Contact( #TB1AlmSupp )
      Coil( #SS_Warning.StopBefor )
   END_RUNG
   // the same network as SCL:
   #SS_Warning.StopBefor := #SB1ModeStopBefor AND NOT #TB1AlmSupp;
END_REGION

REGION Network 29: Warning - Stop after active
   RUNG wire#powerrail
      Contact( #SB1ModeStopAfter )
      I_Contact( #TB1AlmSupp )
      Coil( #SS_Warning.StopAfter )
   END_RUNG
   // the same network as SCL:
   #SS_Warning.StopAfter := #SB1ModeStopAfter AND NOT #TB1AlmSupp;
END_REGION

REGION Network 30: Warning - Mode Bypass Active
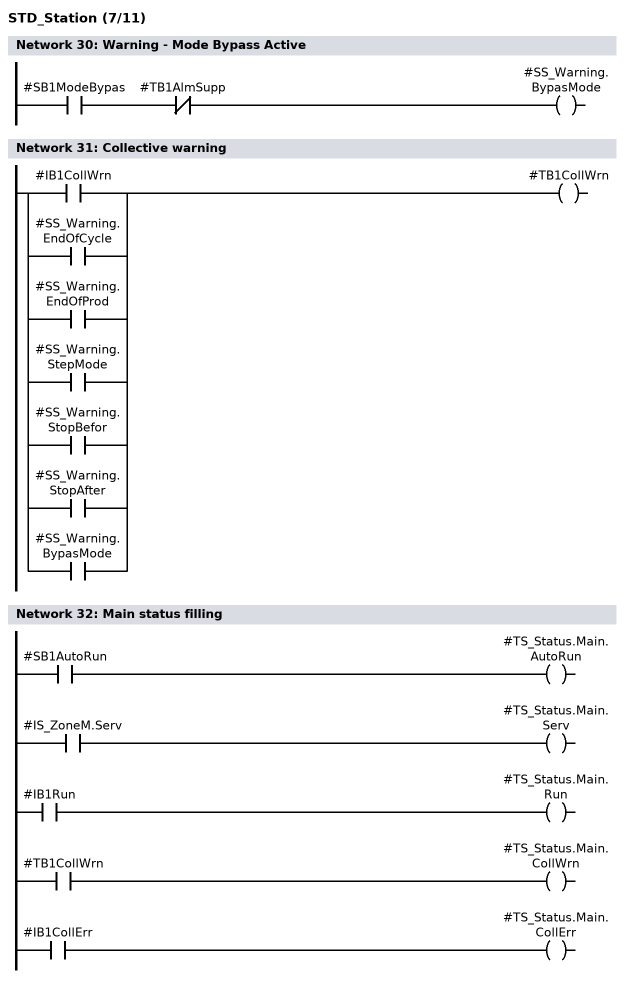
   RUNG wire#powerrail
      Contact( #SB1ModeBypas )
      I_Contact( #TB1AlmSupp )
      Coil( #SS_Warning.BypasMode )
   END_RUNG
   // the same network as SCL:
   #SS_Warning.BypasMode := #SB1ModeBypas AND NOT #TB1AlmSupp;
END_REGION

REGION Network 31: Collective warning
   RUNG wire#powerrail
      Contact( #IB1CollWrn )
      wire#w1
      Coil( #TB1CollWrn )
   END_RUNG
   RUNG wire#powerrail
      Contact( #SS_Warning.EndOfCycle )
   END_RUNG wire#w1
   RUNG wire#powerrail
      Contact( #SS_Warning.EndOfProd )
   END_RUNG wire#w1
   RUNG wire#powerrail
      Contact( #SS_Warning.StepMode )
   END_RUNG wire#w1
   RUNG wire#powerrail
      Contact( #SS_Warning.StopBefor )
   END_RUNG wire#w1
   RUNG wire#powerrail
      Contact( #SS_Warning.StopAfter )
   END_RUNG wire#w1
   RUNG wire#powerrail
      Contact( #SS_Warning.BypasMode )
   END_RUNG wire#w1
   // the same network as SCL:
   #TB1CollWrn := #IB1CollWrn OR #SS_Warning.EndOfCycle OR #SS_Warning.EndOfProd OR #SS_Warning.StepMode OR #SS_Warning.StopBefor OR #SS_Warning.StopAfter OR #SS_Warning.BypasMode;
END_REGION

REGION Network 32: Main status filling
   RUNG wire#powerrail
      Contact( #SB1AutoRun )
      Coil( #TS_Status.Main.AutoRun )
   END_RUNG
   RUNG wire#powerrail
      Contact( #IS_ZoneM.Serv )
      Coil( #TS_Status.Main.Serv )
   END_RUNG
   RUNG wire#powerrail
      Contact( #IB1Run )
      Coil( #TS_Status.Main.Run )
   END_RUNG
   RUNG wire#powerrail
      Contact( #TB1CollWrn )
      Coil( #TS_Status.Main.CollWrn )
   END_RUNG
   RUNG wire#powerrail
      Contact( #IB1CollErr )
      Coil( #TS_Status.Main.CollErr )
   END_RUNG
   // the same network as SCL:
   #TS_Status.Main.AutoRun := #SB1AutoRun;
   #TS_Status.Main.Serv := #IS_ZoneM.Serv;
   #TS_Status.Main.Run := #IB1Run;
   #TS_Status.Main.CollWrn := #TB1CollWrn;
   #TS_Status.Main.CollErr := #IB1CollErr;
END_REGION

REGION Network 33: Specific status filling
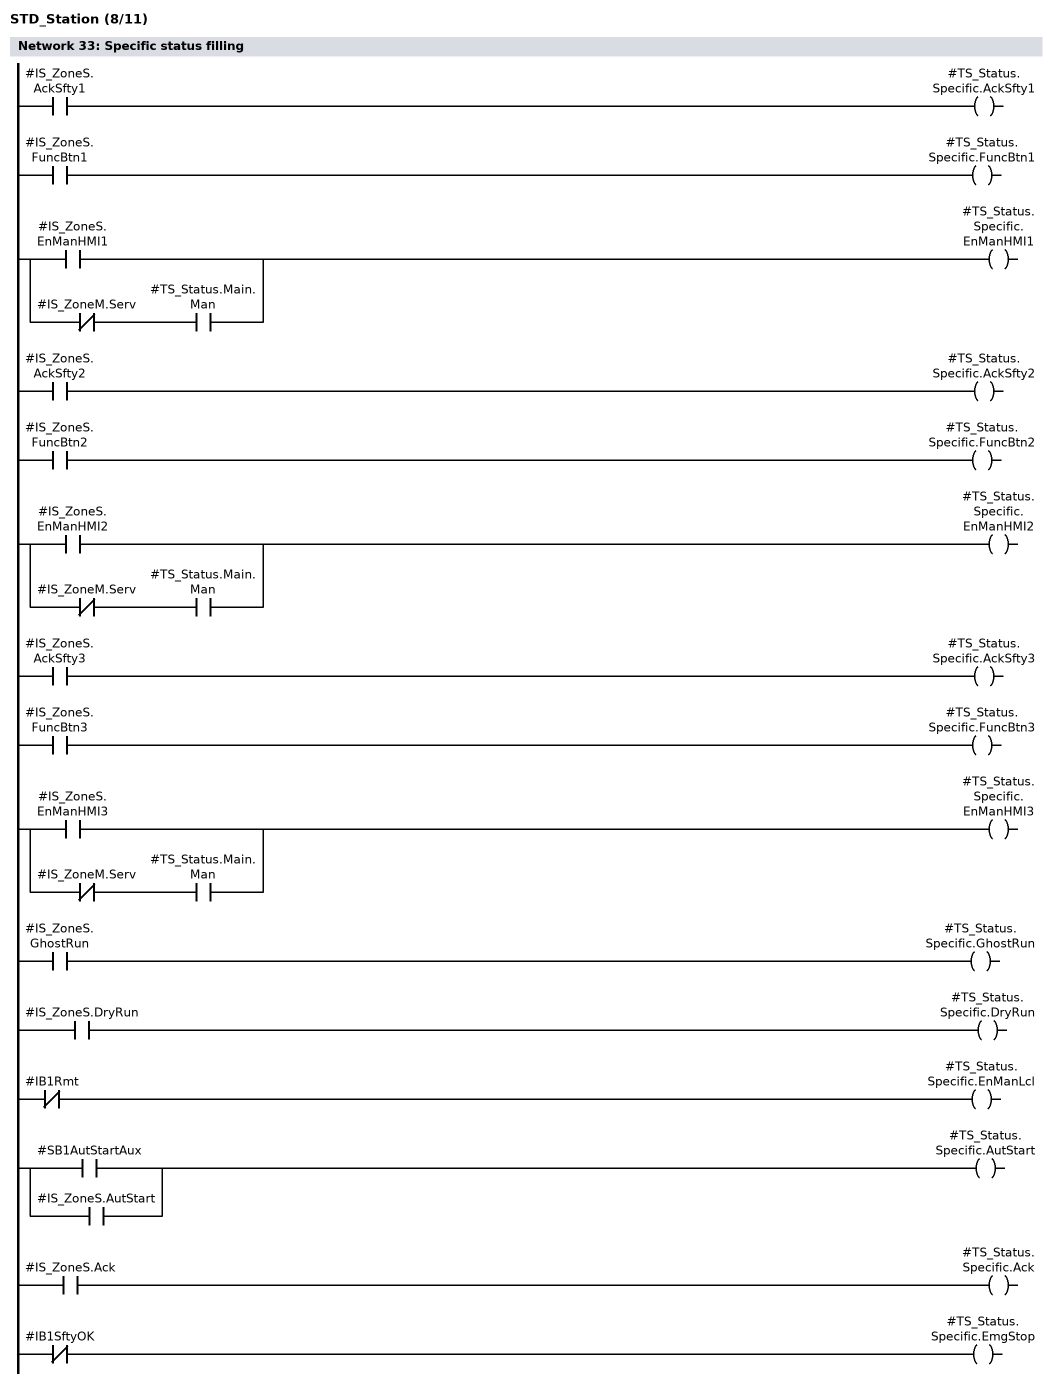
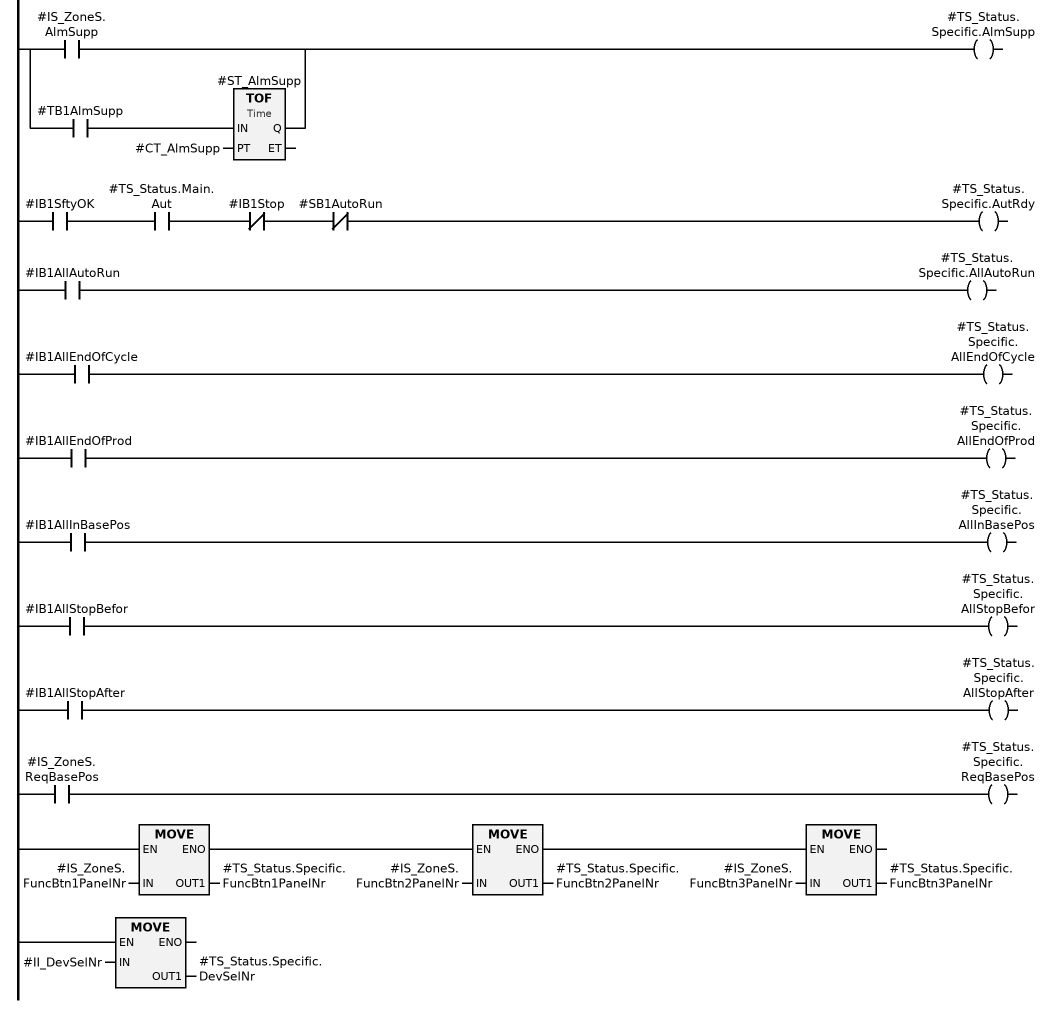
   RUNG wire#powerrail
      Contact( #IS_ZoneS.AckSfty1 )
      Coil( #TS_Status.Specific.AckSfty1 )
   END_RUNG
   RUNG wire#powerrail
      Contact( #IS_ZoneS.FuncBtn1 )
      Coil( #TS_Status.Specific.FuncBtn1 )
   END_RUNG
   RUNG wire#powerrail
      Contact( #IS_ZoneS.EnManHMI1 )
      wire#w1
      Coil( #TS_Status.Specific.EnManHMI1 )
   END_RUNG
   RUNG wire#powerrail
      I_Contact( #IS_ZoneM.Serv )
      Contact( #TS_Status.Main.Man )
   END_RUNG wire#w1
   RUNG wire#powerrail
      Contact( #IS_ZoneS.AckSfty2 )
      Coil( #TS_Status.Specific.AckSfty2 )
   END_RUNG
   RUNG wire#powerrail
      Contact( #IS_ZoneS.FuncBtn2 )
      Coil( #TS_Status.Specific.FuncBtn2 )
   END_RUNG
   RUNG wire#powerrail
      Contact( #IS_ZoneS.EnManHMI2 )
      wire#w2
      Coil( #TS_Status.Specific.EnManHMI2 )
   END_RUNG
   RUNG wire#powerrail
      I_Contact( #IS_ZoneM.Serv )
      Contact( #TS_Status.Main.Man )
   END_RUNG wire#w2
   RUNG wire#powerrail
      Contact( #IS_ZoneS.AckSfty3 )
      Coil( #TS_Status.Specific.AckSfty3 )
   END_RUNG
   RUNG wire#powerrail
      Contact( #IS_ZoneS.FuncBtn3 )
      Coil( #TS_Status.Specific.FuncBtn3 )
   END_RUNG
   RUNG wire#powerrail
      Contact( #IS_ZoneS.EnManHMI3 )
      wire#w3
      Coil( #TS_Status.Specific.EnManHMI3 )
   END_RUNG
   RUNG wire#powerrail
      I_Contact( #IS_ZoneM.Serv )
      Contact( #TS_Status.Main.Man )
   END_RUNG wire#w3
   RUNG wire#powerrail
      Contact( #IS_ZoneS.GhostRun )
      Coil( #TS_Status.Specific.GhostRun )
   END_RUNG
   RUNG wire#powerrail
      Contact( #IS_ZoneS.DryRun )
      Coil( #TS_Status.Specific.DryRun )
   END_RUNG
   RUNG wire#powerrail
      I_Contact( #IB1Rmt )
      Coil( #TS_Status.Specific.EnManLcl )
   END_RUNG
   RUNG wire#powerrail
      Contact( #SB1AutStartAux )
      wire#w4
      Coil( #TS_Status.Specific.AutStart )
   END_RUNG
   RUNG wire#powerrail
      Contact( #IS_ZoneS.AutStart )
   END_RUNG wire#w4
   RUNG wire#powerrail
      Contact( #IS_ZoneS.Ack )
      Coil( #TS_Status.Specific.Ack )
   END_RUNG
   RUNG wire#powerrail
      I_Contact( #IB1SftyOK )
      Coil( #TS_Status.Specific.EmgStop )
   END_RUNG
   RUNG wire#powerrail
      Contact( #IS_ZoneS.AlmSupp )
      wire#w5
      Coil( #TS_Status.Specific.AlmSupp )
   END_RUNG
   RUNG wire#powerrail
      Contact( #TB1AlmSupp )
      { S7_Templates := "time_type := Time" } #ST_AlmSupp.TOF(pt := #CT_AlmSupp, et =>)
   END_RUNG wire#w5
   RUNG wire#powerrail
      Contact( #IB1SftyOK )
      Contact( #TS_Status.Main.Aut )
      I_Contact( #IB1Stop )
      I_Contact( #SB1AutoRun )
      Coil( #TS_Status.Specific.AutRdy )
   END_RUNG
   RUNG wire#powerrail
      Contact( #IB1AllAutoRun )
      Coil( #TS_Status.Specific.AllAutoRun )
   END_RUNG
   RUNG wire#powerrail
      Contact( #IB1AllEndOfCycle )
      Coil( #TS_Status.Specific.AllEndOfCycle )
   END_RUNG
   RUNG wire#powerrail
      Contact( #IB1AllEndOfProd )
      Coil( #TS_Status.Specific.AllEndOfProd )
   END_RUNG
   RUNG wire#powerrail
      Contact( #IB1AllInBasePos )
      Coil( #TS_Status.Specific.AllInBasePos )
   END_RUNG
   RUNG wire#powerrail
      Contact( #IB1AllStopBefor )
      Coil( #TS_Status.Specific.AllStopBefor )
   END_RUNG
   RUNG wire#powerrail
      Contact( #IB1AllStopAfter )
      Coil( #TS_Status.Specific.AllStopAfter )
   END_RUNG
   RUNG wire#powerrail
      Contact( #IS_ZoneS.ReqBasePos )
      Coil( #TS_Status.Specific.ReqBasePos )
   END_RUNG
   RUNG wire#powerrail
      { S7_GenerateENO := "TRUE" } Move(in := #IS_ZoneS.FuncBtn1PanelNr, out1 => #TS_Status.Specific.FuncBtn1PanelNr)
      { S7_GenerateENO := "TRUE" } Move(in := #IS_ZoneS.FuncBtn2PanelNr, out1 => #TS_Status.Specific.FuncBtn2PanelNr)
      { S7_GenerateENO := "TRUE" } Move(in := #IS_ZoneS.FuncBtn3PanelNr, out1 => #TS_Status.Specific.FuncBtn3PanelNr)
   END_RUNG
   RUNG wire#powerrail
      { S7_GenerateENO := "TRUE" } Move(in := #II_DevSelNr, out1 => #TS_Status.Specific.DevSelNr)
   END_RUNG
   // the same network as SCL:
   // ENO of a box is taken as its EN; it also drops when the box reports an error
   #TS_Status.Specific.AckSfty1 := #IS_ZoneS.AckSfty1;
   #TS_Status.Specific.FuncBtn1 := #IS_ZoneS.FuncBtn1;
   #TS_Status.Specific.EnManHMI1 := #IS_ZoneS.EnManHMI1 OR (NOT #IS_ZoneM.Serv AND #TS_Status.Main.Man);
   #TS_Status.Specific.AckSfty2 := #IS_ZoneS.AckSfty2;
   #TS_Status.Specific.FuncBtn2 := #IS_ZoneS.FuncBtn2;
   #TS_Status.Specific.EnManHMI2 := #IS_ZoneS.EnManHMI2 OR (NOT #IS_ZoneM.Serv AND #TS_Status.Main.Man);
   #TS_Status.Specific.AckSfty3 := #IS_ZoneS.AckSfty3;
   #TS_Status.Specific.FuncBtn3 := #IS_ZoneS.FuncBtn3;
   #TS_Status.Specific.EnManHMI3 := #IS_ZoneS.EnManHMI3 OR (NOT #IS_ZoneM.Serv AND #TS_Status.Main.Man);
   #TS_Status.Specific.GhostRun := #IS_ZoneS.GhostRun;
   #TS_Status.Specific.DryRun := #IS_ZoneS.DryRun;
   #TS_Status.Specific.EnManLcl := NOT #IB1Rmt;
   #TS_Status.Specific.AutStart := #SB1AutStartAux OR #IS_ZoneS.AutStart;
   #TS_Status.Specific.Ack := #IS_ZoneS.Ack;
   #TS_Status.Specific.EmgStop := NOT #IB1SftyOK;
   #ST_AlmSupp.TOF(IN := #TB1AlmSupp, PT := #CT_AlmSupp);
   #TS_Status.Specific.AlmSupp := #IS_ZoneS.AlmSupp OR #ST_AlmSupp.Q;
   #TS_Status.Specific.AutRdy := #IB1SftyOK AND #TS_Status.Main.Aut AND NOT #IB1Stop AND NOT #SB1AutoRun;
   #TS_Status.Specific.AllAutoRun := #IB1AllAutoRun;
   #TS_Status.Specific.AllEndOfCycle := #IB1AllEndOfCycle;
   #TS_Status.Specific.AllEndOfProd := #IB1AllEndOfProd;
   #TS_Status.Specific.AllInBasePos := #IB1AllInBasePos;
   #TS_Status.Specific.AllStopBefor := #IB1AllStopBefor;
   #TS_Status.Specific.AllStopAfter := #IB1AllStopAfter;
   #TS_Status.Specific.ReqBasePos := #IS_ZoneS.ReqBasePos;
   #TS_Status.Specific.FuncBtn1PanelNr := #IS_ZoneS.FuncBtn1PanelNr;
   #TS_Status.Specific.FuncBtn2PanelNr := #IS_ZoneS.FuncBtn2PanelNr;
   #TS_Status.Specific.FuncBtn3PanelNr := #IS_ZoneS.FuncBtn3PanelNr;
   #TS_Status.Specific.DevSelNr := #II_DevSelNr;
END_REGION

REGION Network 34: Reset commands
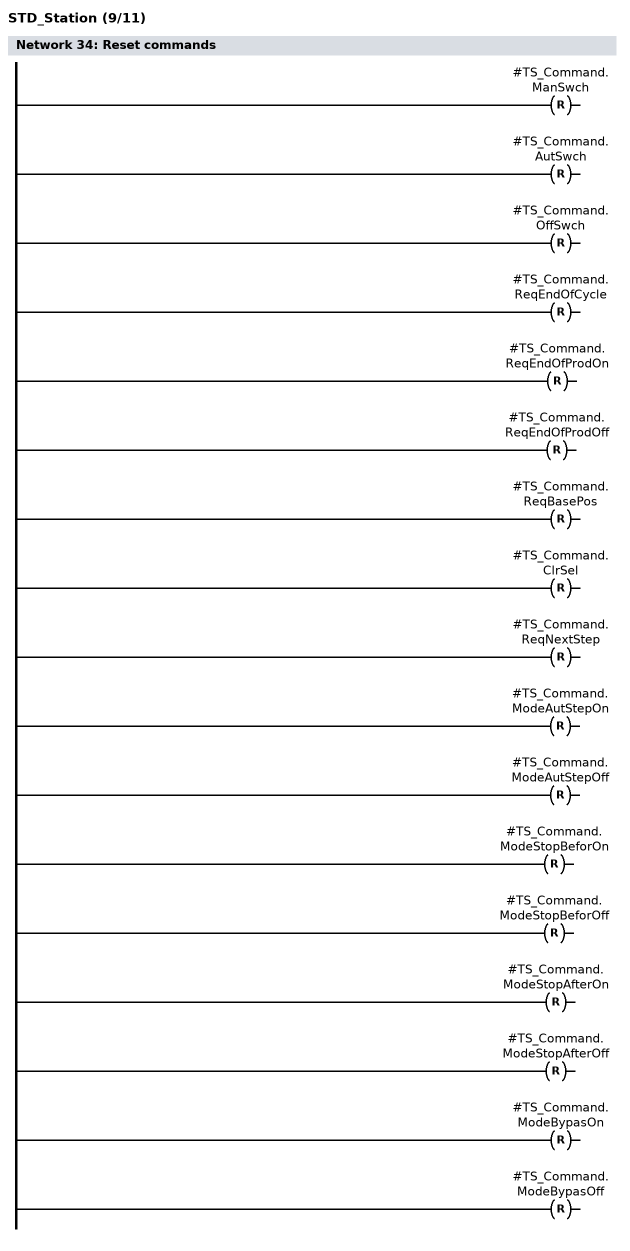
   RUNG wire#powerrail
      R_Coil( #TS_Command.ManSwch )
   END_RUNG
   RUNG wire#powerrail
      R_Coil( #TS_Command.AutSwch )
   END_RUNG
   RUNG wire#powerrail
      R_Coil( #TS_Command.OffSwch )
   END_RUNG
   RUNG wire#powerrail
      R_Coil( #TS_Command.ReqEndOfCycle )
   END_RUNG
   RUNG wire#powerrail
      R_Coil( #TS_Command.ReqEndOfProdOn )
   END_RUNG
   RUNG wire#powerrail
      R_Coil( #TS_Command.ReqEndOfProdOff )
   END_RUNG
   RUNG wire#powerrail
      R_Coil( #TS_Command.ReqBasePos )
   END_RUNG
   RUNG wire#powerrail
      R_Coil( #TS_Command.ClrSel )
   END_RUNG
   RUNG wire#powerrail
      R_Coil( #TS_Command.ReqNextStep )
   END_RUNG
   RUNG wire#powerrail
      R_Coil( #TS_Command.ModeAutStepOn )
   END_RUNG
   RUNG wire#powerrail
      R_Coil( #TS_Command.ModeAutStepOff )
   END_RUNG
   RUNG wire#powerrail
      R_Coil( #TS_Command.ModeStopBeforOn )
   END_RUNG
   RUNG wire#powerrail
      R_Coil( #TS_Command.ModeStopBeforOff )
   END_RUNG
   RUNG wire#powerrail
      R_Coil( #TS_Command.ModeStopAfterOn )
   END_RUNG
   RUNG wire#powerrail
      R_Coil( #TS_Command.ModeStopAfterOff )
   END_RUNG
   RUNG wire#powerrail
      R_Coil( #TS_Command.ModeBypasOn )
   END_RUNG
   RUNG wire#powerrail
      R_Coil( #TS_Command.ModeBypasOff )
   END_RUNG
   // the same network as SCL:
   #TS_Command.ManSwch := FALSE;
   #TS_Command.AutSwch := FALSE;
   #TS_Command.OffSwch := FALSE;
   #TS_Command.ReqEndOfCycle := FALSE;
   #TS_Command.ReqEndOfProdOn := FALSE;
   #TS_Command.ReqEndOfProdOff := FALSE;
   #TS_Command.ReqBasePos := FALSE;
   #TS_Command.ClrSel := FALSE;
   #TS_Command.ReqNextStep := FALSE;
   #TS_Command.ModeAutStepOn := FALSE;
   #TS_Command.ModeAutStepOff := FALSE;
   #TS_Command.ModeStopBeforOn := FALSE;
   #TS_Command.ModeStopBeforOff := FALSE;
   #TS_Command.ModeStopAfterOn := FALSE;
   #TS_Command.ModeStopAfterOff := FALSE;
   #TS_Command.ModeBypasOn := FALSE;
   #TS_Command.ModeBypasOff := FALSE;
END_REGION

REGION Network 35: Alarms - copy to structure
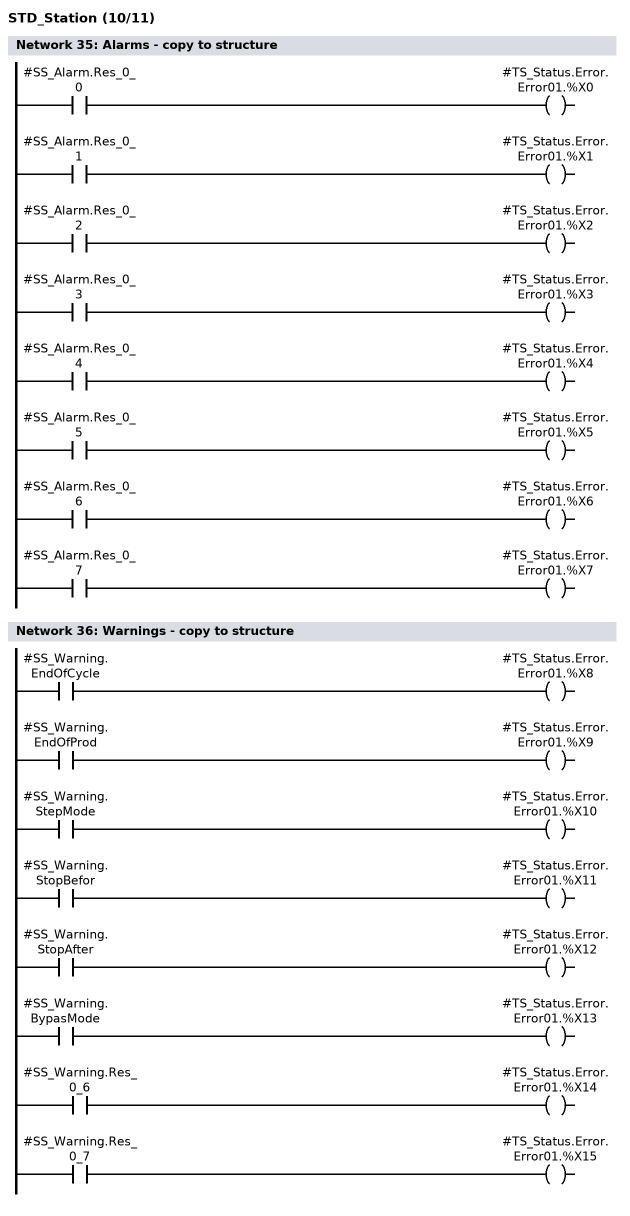
   RUNG wire#powerrail
      Contact( #SS_Alarm.Res_0_0 )
      Coil( #TS_Status.Error.Error01.%X0 )
   END_RUNG
   RUNG wire#powerrail
      Contact( #SS_Alarm.Res_0_1 )
      Coil( #TS_Status.Error.Error01.%X1 )
   END_RUNG
   RUNG wire#powerrail
      Contact( #SS_Alarm.Res_0_2 )
      Coil( #TS_Status.Error.Error01.%X2 )
   END_RUNG
   RUNG wire#powerrail
      Contact( #SS_Alarm.Res_0_3 )
      Coil( #TS_Status.Error.Error01.%X3 )
   END_RUNG
   RUNG wire#powerrail
      Contact( #SS_Alarm.Res_0_4 )
      Coil( #TS_Status.Error.Error01.%X4 )
   END_RUNG
   RUNG wire#powerrail
      Contact( #SS_Alarm.Res_0_5 )
      Coil( #TS_Status.Error.Error01.%X5 )
   END_RUNG
   RUNG wire#powerrail
      Contact( #SS_Alarm.Res_0_6 )
      Coil( #TS_Status.Error.Error01.%X6 )
   END_RUNG
   RUNG wire#powerrail
      Contact( #SS_Alarm.Res_0_7 )
      Coil( #TS_Status.Error.Error01.%X7 )
   END_RUNG
   // the same network as SCL:
   #TS_Status.Error.Error01.%X0 := #SS_Alarm.Res_0_0;
   #TS_Status.Error.Error01.%X1 := #SS_Alarm.Res_0_1;
   #TS_Status.Error.Error01.%X2 := #SS_Alarm.Res_0_2;
   #TS_Status.Error.Error01.%X3 := #SS_Alarm.Res_0_3;
   #TS_Status.Error.Error01.%X4 := #SS_Alarm.Res_0_4;
   #TS_Status.Error.Error01.%X5 := #SS_Alarm.Res_0_5;
   #TS_Status.Error.Error01.%X6 := #SS_Alarm.Res_0_6;
   #TS_Status.Error.Error01.%X7 := #SS_Alarm.Res_0_7;
END_REGION

REGION Network 36: Warnings - copy to structure
   RUNG wire#powerrail
      Contact( #SS_Warning.EndOfCycle )
      Coil( #TS_Status.Error.Error01.%X8 )
   END_RUNG
   RUNG wire#powerrail
      Contact( #SS_Warning.EndOfProd )
      Coil( #TS_Status.Error.Error01.%X9 )
   END_RUNG
   RUNG wire#powerrail
      Contact( #SS_Warning.StepMode )
      Coil( #TS_Status.Error.Error01.%X10 )
   END_RUNG
   RUNG wire#powerrail
      Contact( #SS_Warning.StopBefor )
      Coil( #TS_Status.Error.Error01.%X11 )
   END_RUNG
   RUNG wire#powerrail
      Contact( #SS_Warning.StopAfter )
      Coil( #TS_Status.Error.Error01.%X12 )
   END_RUNG
   RUNG wire#powerrail
      Contact( #SS_Warning.BypasMode )
      Coil( #TS_Status.Error.Error01.%X13 )
   END_RUNG
   RUNG wire#powerrail
      Contact( #SS_Warning.Res_0_6 )
      Coil( #TS_Status.Error.Error01.%X14 )
   END_RUNG
   RUNG wire#powerrail
      Contact( #SS_Warning.Res_0_7 )
      Coil( #TS_Status.Error.Error01.%X15 )
   END_RUNG
   // the same network as SCL:
   #TS_Status.Error.Error01.%X8 := #SS_Warning.EndOfCycle;
   #TS_Status.Error.Error01.%X9 := #SS_Warning.EndOfProd;
   #TS_Status.Error.Error01.%X10 := #SS_Warning.StepMode;
   #TS_Status.Error.Error01.%X11 := #SS_Warning.StopBefor;
   #TS_Status.Error.Error01.%X12 := #SS_Warning.StopAfter;
   #TS_Status.Error.Error01.%X13 := #SS_Warning.BypasMode;
   #TS_Status.Error.Error01.%X14 := #SS_Warning.Res_0_6;
   #TS_Status.Error.Error01.%X15 := #SS_Warning.Res_0_7;
END_REGION

REGION Network 37: Copy to output structure
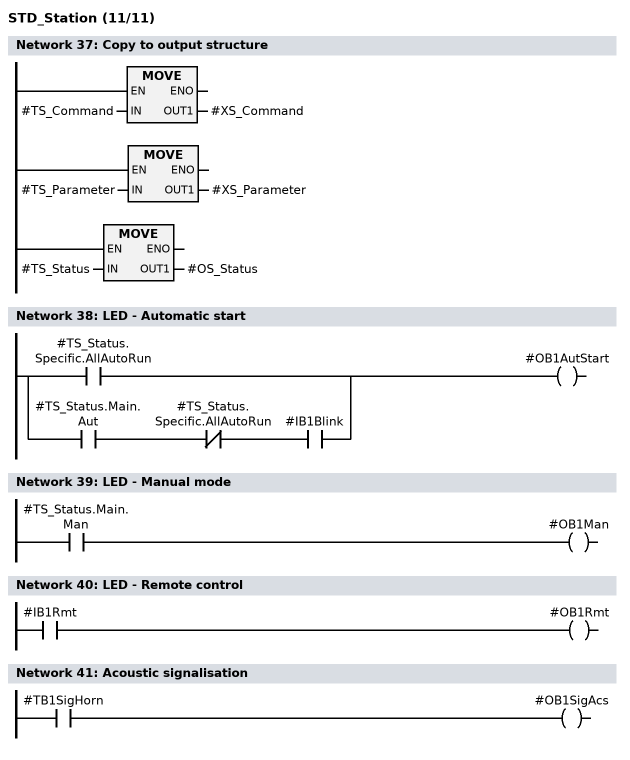
   RUNG wire#powerrail
      { S7_GenerateENO := "TRUE" } Move(in := #TS_Command, out1 => #XS_Command)
   END_RUNG
   RUNG wire#powerrail
      { S7_GenerateENO := "TRUE" } Move(in := #TS_Parameter, out1 => #XS_Parameter)
   END_RUNG
   RUNG wire#powerrail
      { S7_GenerateENO := "TRUE" } Move(in := #TS_Status, out1 => #OS_Status)
   END_RUNG
   // the same network as SCL:
   #XS_Command := #TS_Command;
   #XS_Parameter := #TS_Parameter;
   #OS_Status := #TS_Status;
END_REGION

REGION Network 38: LED - Automatic start
   RUNG wire#powerrail
      Contact( #TS_Status.Specific.AllAutoRun )
      wire#w1
      Coil( #OB1AutStart )
   END_RUNG
   RUNG wire#powerrail
      Contact( #TS_Status.Main.Aut )
      I_Contact( #TS_Status.Specific.AllAutoRun )
      Contact( #IB1Blink )
   END_RUNG wire#w1
   // the same network as SCL:
   #OB1AutStart := #TS_Status.Specific.AllAutoRun OR (#TS_Status.Main.Aut AND NOT #TS_Status.Specific.AllAutoRun AND #IB1Blink);
END_REGION

REGION Network 39: LED - Manual mode
   RUNG wire#powerrail
      Contact( #TS_Status.Main.Man )
      Coil( #OB1Man )
   END_RUNG
   // the same network as SCL:
   #OB1Man := #TS_Status.Main.Man;
END_REGION

REGION Network 40: LED - Remote control
   RUNG wire#powerrail
      Contact( #IB1Rmt )
      Coil( #OB1Rmt )
   END_RUNG
   // the same network as SCL:
   #OB1Rmt := #IB1Rmt;
END_REGION

REGION Network 41: Acoustic signalisation
   RUNG wire#powerrail
      Contact( #TB1SigHorn )
      Coil( #OB1SigAcs )
   END_RUNG
   // the same network as SCL:
   #OB1SigAcs := #TB1SigHorn;
END_REGION
END_FUNCTION_BLOCK
